DATA_BLOCK "DB_maXYmosNC1"
VAR
  ProgNo : Int;
  SelectSeq : Int;
  ZeroX : Bool;
  SetXRef : Bool;
  Homing : Bool;
  StartCycle : Bool;
  ContinueSeq : Bool;
  JogPos : Bool;
  JogNeg : Bool;
  JogPosActive : Bool;
  JogNegActive : Bool;
  SpareByte : Array[0..67] of Byte;
  InputMessages : STRUCT
    StatusBits : STRUCT
      "MIRROR-START" : Bool;
      "MIRROR-TARE-Y" : Bool;
      "MIRROR-ZERO X" : Bool;
      "MIRROR-STEST-X" : Bool;
      "MIRROR-STEST-Y" : Bool;
      "ReservedBit000.5" : Bool;
      "MASTER-MEAS" : Bool;
      "INC-ZERO" : Bool;
      "ReservedBit001.0" : Bool;
      "MIRROR-ACK-ADMIN" : Bool;
      "ReservedBit001.2" : Bool;
      "MIRROR-ACCESS" : Bool;
      AUTO : Bool;
      "STAT-RESET" : Bool;
      "STAT-DISABLE" : Bool;
      "TARE-EXTENDED-Y" : Bool;
      MP : Byte;
      "ReservedBit003.0" : Bool;
      "ReservedBit003.1" : Bool;
      "RESET-SN-GENERATOR" : Bool;
      "ReservedBit003.3" : Bool;
      "ReservedBit003.4" : Bool;
      "BREAKETEST-ACTIVE" : Bool;
      "ReservedBit003.6" : Bool;
      "ReservedBit003.7" : Bool;
      UNI : Byte;
      ReservedByte005 : Byte;
      READY : Bool;
      "OK-TOTAL" : Bool;
      "NOK-TOTAL" : Bool;
      "NO-PASS" : Bool;
      "ReservedBit006.4" : Bool;
      "ReservedBit006.5" : Bool;
      WARN : Bool;
      ALARM : Bool;
      S1 : Bool;
      S2 : Bool;
      "ReservedBit007.2" : Bool;
      "ReservedBit007.3" : Bool;
      "ReservedBit007.4" : Bool;
      "ReservedBit007.5" : Bool;
      "ReservedBit007.6" : Bool;
      "ReservedBit007.7" : Bool;
      "O-UNI" : Byte;
      "DRIVE-ENABLE" : Bool;
      "RUN-SEQUENCE" : Bool;
      "DRIVE-TO-HOMEPOS" : Bool;
      "DRIVE-TO-REFPOS" : Bool;
      "JOG-FW" : Bool;
      "JOG-BW" : Bool;
      "WAIT-REQUEST" : Bool;
      "BRAKETEST-DONE" : Bool;
      "SEQUENCE-STOPPED" : Bool;
      "SEQUENCE-END" : Bool;
      "ONLINE-EO-NOK" : Bool;
      "EXT-STOP" : Bool;
      "SEQUENCE-ERROR" : Bool;
      "DRIVE-ENABLED" : Bool;
      "HOMEPOS-REACHED" : Bool;
      "REFPOS-REACHED" : Bool;
      STANDSTILL : Bool;
      "BRAKETEST-REQ" : Bool;
      "SERVO-WARN" : Bool;
      "SERVO-ERROR" : Bool;
      "SMES-ACTIVE" : Bool;
      "SMST2-ACTIVE" : Bool;
      "SMM1-ACTIVE" : Bool;
      "USER-MODE-ACTIVE" : Bool;
      SEQUENCE : Byte;
      "LABEL-ID" : Byte;
      "CFG-MP" : Byte;
      "ReservedBit015.0" : Bool;
      "ReservedBit015.1" : Bool;
      "ReservedBit015.2" : Bool;
      "ReservedBit015.3" : Bool;
      "ReservedBit015.4" : Bool;
      "ReservedBit015.5" : Bool;
      "ReservedBit015.6" : Bool;
      "GLOBAL-CFG-MP" : Bool;
      "MIRRIR-CFG-ADR" : Byte;
      "MIRRIR-CFG-LENGTH" : Byte;
      "SELECT-PAGE" : Byte;
      "TRANSMISSION-FAULT" : Bool;
      ACK : Bool;
      "DEVICE-AVAILABLE" : Bool;
      "ReservedBit019.3" : Bool;
      "CHANGEDSELECTED-MP" : Bool;
      "ReservedBit019.5" : Bool;
      "CHANGED--GLOBAL" : Bool;
      "BACKUP-REQUEST" : Bool;
    END_STRUCT;
    FreelyArea : STRUCT
      XEncRefValue : Real;
      CurValueX_1 : Real;
      CurValueX_2 : Real;
      CurValueY : Real;
      SerialNnmber : Array[36..85] of Byte;
      "pvCurveXMIN-X" : Real;
      "pvCurveXMAX-X" : Real;
      "pvCurveYMIN-Y" : Real;
      "pvCurveYMAX-Y" : Real;
      PressData : Array[86..203] of Byte;
    END_STRUCT;
  END_STRUCT;
  OutputMessages : STRUCT
    ControlBits : STRUCT
      START : Bool;
      "TARE-Y" : Bool;
      "ZERO X" : Bool;
      "STEST-X" : Bool;
      "STEST-Y" : Bool;
      "ReservedBit000.5" : Bool;
      "MASTER-MEAS" : Bool;
      "INC-ZERO" : Bool;
      "ReservedBit001.0" : Bool;
      "ACK-ADMIN" : Bool;
      "ReservedBit001.2" : Bool;
      ACCESS : Bool;
      AUTO : Bool;
      "STAT-RESET" : Bool;
      "STAT-DISABLE" : Bool;
      "TARE-EXTENDED-Y" : Bool;
      MP : Byte;
      "ReservedBit003.0" : Bool;
      "ReservedBit003.1" : Bool;
      "RESET-SN-GENERATOR" : Bool;
      "ReservedBit003.3" : Bool;
      "ReservedBit003.4" : Bool;
      "ReservedBit003.5" : Bool;
      "ReservedBit003.6" : Bool;
      "ReservedBit003.7" : Bool;
      UNI : Byte;
      ReservedByte005 : Byte;
      ReservedByte006 : Byte;
      ReservedByte007 : Byte;
      ReservedByte008 : Byte;
      "DRIVE-ENABLE" : Bool;
      "RUN-SEQUENCE" : Bool;
      "DRIVE-TO-HOMEPOS" : Bool;
      "DRIVE-TO-REFPOS" : Bool;
      "JOG-FW" : Bool;
      "JOG-BW" : Bool;
      "CONTNUEFROM-WAIT" : Bool;
      "MANUAL-BRAKETEST" : Bool;
      "ReservedBit010.0" : Bool;
      "ReservedBit010.1" : Bool;
      "ReservedBit010.2" : Bool;
      "SEQ-EXT-STOP-REQ" : Bool;
      "ReservedBit010.4" : Bool;
      "ReservedBit010.5" : Bool;
      "ReservedBit010.6" : Bool;
      "ReservedBit010.7" : Bool;
      ReservedByte011 : Byte;
      "CURRENT SEQUENCE" : Byte;
      ReservedByte013 : Byte;
      "CFG-MP" : Byte;
      "ReservedBit015.0" : Bool;
      "ReservedBit015.1" : Bool;
      "ReservedBit015.2" : Bool;
      "ReservedBit015.3" : Bool;
      "ReservedBit015.4" : Bool;
      "ReservedBit015.5" : Bool;
      "ReservedBit015.6" : Bool;
      "GLOBAL-CFG-MP" : Bool;
      "CFG-ADDRESS" : Byte;
      "CFG-LENGTH" : Byte;
      "SELECT-PAGE" : Byte;
      "SAVE-TO-MP" : Bool;
      STROBE : Bool;
      "ReservedBit019.2" : Bool;
      "ReservedBit019.3" : Bool;
      "RESET-CHANGED-SELECTED-MP" : Bool;
      "ReservedBit019.5" : Bool;
      "RESET-CHANGEDGLOBAL" : Bool;
      "BACKUP-REQUEST" : Bool;
    END_STRUCT;
    FreelyArea : STRUCT
      XEncRefValue : Real;
      JogSpeed : Real;
      JogMaxForce : Real;
      CalibForce : Real;
      SerialNnmber : Array[36..85] of Byte;
      PressData : Array[86..219] of Byte;
    END_STRUCT;
  END_STRUCT;
  Info : STRUCT
    ProgNo : Byte;
    SelectSeq : Byte;
    SelectPage : Byte;
    CfgAddress : Byte;
    CfgLength : Byte;
    Cancel : Bool;
    ContinueSeq : Bool;
  END_STRUCT;
  SetXRefRise : Bool;
  JogRise : Bool;
  HomingRise : Bool;
  StartCycleRise : Bool;
  FltQuitRise : Bool;
  SetXRefOld : Bool;
  JogOld : Bool;
  HomingOld : Bool;
  StartCycleOld : Bool;
  FltQuitOld : Bool;
  SetXRefAct : Bool;
  JogAct : Bool;
  HomeAct : Bool;
  CycleAct : Bool;
  OrderCount : Int;
  Index : Int;
  Step : Array[1..5] of Int;
  Ref_Timer_IN : Bool;
  JogTimer_IN : Bool;
  HomeTimer_IN : Bool;
  SeqTimer_IN : Bool;
  HomeTime : Time;
  SeqTime : Time;
  Ref_Timer : TON_TIME;
  Jog_Timer : TON_TIME;
  Home_Timer : TON_TIME;
  Seq_Timer : TON_TIME;
END_VAR
BEGIN
END_DATA_BLOCK
